{attribute 'GeneratedUsingTerminal: EJ2522-0000-0022'}
{attribute addProperty BoxType "EJ2522-0000-0022"}
{attribute addProperty Id "Set_counter_doneBOOL1Counter_underflowBOOL1Counter_overflowBOOL1Sync_errorBOOL1TxPDO_StateBOOL1TxPDO_ToggleBOOL1"}
{attribute addProperty CRC "1893737464"}
{attribute addProperty Size "6"}
TYPE Status_70E023F8 :
STRUCT
	{attribute addProperty Name "Set_counter_done"}
	Set_counter_done : BOOL;
	{attribute addProperty Name "Counter_underflow"}
	Counter_underflow : BOOL;
	{attribute addProperty Name "Counter_overflow"}
	Counter_overflow : BOOL;
	{attribute addProperty Name "Sync_error"}
	Sync_error : BOOL;
	{attribute addProperty Name "TxPDO_State"}
	TxPDO_State : BOOL;
	{attribute addProperty Name "TxPDO_Toggle"}
	TxPDO_Toggle : BOOL;
END_STRUCT
END_TYPE

(* stored: Version 1.2.0.0, ProductVersion 3.1.4024.9
   DUT Status_70E023F8: Id {921d5d52-b373-4f78-826d-6e08d9d0498b} *)
